// TIA Portal project "1.简易传送带控制程序-1200_V17" (V17)
// Vorlageprojekt für das Buch mit Zielsystem S7-1200

(* hardware
DEVICE "S7-1200-Station_1"  S7-1200 Station
   slot 0: "Baugruppenträger_0"  Rack  V1.0
   slot 1: "PLC_1"  CPU 1214C DC/DC/Rly  6ES7 214-1HG40-0XB0  V4.4
*)

// ===== PLC "PLC_1"  CPU 1214C DC/DC/Rly =====

VAR_GLOBAL   // PLC tag table "Standard-Variablentabelle"
   "运行指示" AT %A0.0 : Bool;
   "启动按钮" AT %E0.0 : Bool;
   "停止按钮" AT %E0.1 : Bool;
   "电机运行标志位" AT %M10.0 : Bool;
   "暂停按钮" AT %I0.2 : Bool;
   "电机" AT %Q0.3 : Bool;
   "停止指示" AT %Q0.1 : Bool;
   "暂停指示" AT %Q0.2 : Bool;
END_VAR

FUNCTION "MHJ-PLC-Lab-Function-S71200" : Void   // FC9000, SCL
{ S7_Optimized_Access := 'TRUE' }
VERSION : 0.1
   VAR_TEMP
      rdTimeReturn : Int;
      outputTime : DTL;
      SyncVal : Byte;
      forVal : Int;
      forVal_2 : Int;
      Value : Byte;
   END_VAR
   VAR CONSTANT
      CompVal : Byte := 16#34;
      Value_01 : Byte := 16#11;
      Value_01_DW : DWord := 16#A165_D992;
      Value_02_DW : DWord := 16#58BE_4401;
   END_VAR
BEGIN

   #Value:=PEEK(area := 16#82,
        dbNumber := 0,
        byteOffset := 511);
   #Value := #Value + 1;

   POKE(area := 16#82,
        dbNumber := 0,
        byteOffset := 511,
        value := #Value);

   POKE(area:=16#81,
        dbNumber:=0,
        byteOffset:=1016,
        value:=#Value_01_DW);
   POKE(area := 16#81,
        dbNumber := 0,
        byteOffset := 1020,
        value := #Value_02_DW);

   POKE(area := 16#81,
        dbNumber := 0,
        byteOffset := 511,
        value := B#16#00);

   FOR #forVal := 0 TO 120 DO
       FOR #forVal_2:=0 TO 10 DO
           #rdTimeReturn:=RD_SYS_T(#outputTime);
           #rdTimeReturn := WR_SYS_T(#outputTime);
           #rdTimeReturn := RD_SYS_T(#outputTime);
           #rdTimeReturn := WR_SYS_T(#outputTime);
       END_FOR;
       #SyncVal:= PEEK(area := 16#81,
                      dbNumber := 0,
                      byteOffset := 511);
       IF #SyncVal = #CompVal THEN
          GOTO M_1;
       END_IF;
   END_FOR;
   RETURN;

   M_1:
   POKE(area := 16#81,
        dbNumber := 0,
        byteOffset := 511,
        value := B#16#0);
END_FUNCTION

ORGANIZATION_BLOCK "Main"   // OB1, LAD, ProgramCycle
TITLE = "Main Program Sweep (Cycle)"
{ S7_Optimized_Access := 'TRUE' }
VERSION : 0.1
   VAR_INPUT
      Initial_Call : Bool;   // Initial call of this OB
      Remanence : Bool;   // =True, if remanent data are available
   END_VAR
BEGIN

REGION Network 1
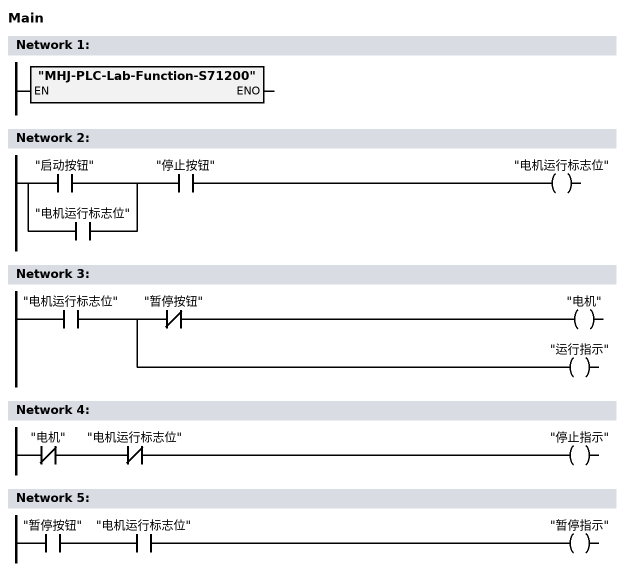
   RUNG wire#powerrail
      "MHJ-PLC-Lab-Function-S71200"()
   END_RUNG
   // the same network as SCL:
   "MHJ-PLC-Lab-Function-S71200"();
END_REGION

REGION Network 2
   RUNG wire#powerrail
      Contact( "启动按钮" )
      wire#w1
      Contact( "停止按钮" )
      Coil( "电机运行标志位" )
   END_RUNG
   RUNG wire#powerrail
      Contact( "电机运行标志位" )
   END_RUNG wire#w1
   // the same network as SCL:
   "电机运行标志位" := ("启动按钮" OR "电机运行标志位") AND "停止按钮";
END_REGION

REGION Network 3
   RUNG wire#powerrail
      Contact( "电机运行标志位" )
      wire#w1
      I_Contact( "暂停按钮" )
      Coil( "电机" )
   END_RUNG
   RUNG wire#w1
      Coil( "运行指示" )
   END_RUNG
   // the same network as SCL:
   "电机" := "电机运行标志位" AND NOT "暂停按钮";
   "运行指示" := "电机运行标志位";
END_REGION

REGION Network 4
   RUNG wire#powerrail
      I_Contact( "电机" )
      I_Contact( "电机运行标志位" )
      Coil( "停止指示" )
   END_RUNG
   // the same network as SCL:
   "停止指示" := NOT "电机" AND NOT "电机运行标志位";
END_REGION

REGION Network 5
   RUNG wire#powerrail
      Contact( "暂停按钮" )
      Contact( "电机运行标志位" )
      Coil( "暂停指示" )
   END_RUNG
   // the same network as SCL:
   "暂停指示" := "暂停按钮" AND "电机运行标志位";
END_REGION
END_ORGANIZATION_BLOCK